FUNCTION_BLOCK FB_Test2 IMPLEMENTS I_BaseString
VAR_INPUT
END_VAR
VAR_OUTPUT
END_VAR
VAR
END_VAR

{warning 'Methodenimplementierung hinzufügen'}
METHOD GetString : STRING
GetString := 'Test 2';
END_METHOD

END_FUNCTION_BLOCK

(* stored: Version 1.1.0.1, ProductVersion 3.1.4024.3
   POU FB_Test2: Id {28e41248-cbcc-4a89-98e5-2bab5b216995}, SpecialFunc None
   Method GetString: Id {e1df74f5-4daf-447a-926f-32a21f571b66} *)
